{attribute 'qualified_only'}
{attribute 'strict'}
{attribute 'to_string'}
TYPE E_CollisionAvoidanceMode :
(
	SINGLE := 0,
	MULTI
);
END_TYPE

(* stored: Version 1.1.0.1
   DUT E_CollisionAvoidanceMode: Id {28e755ba-6279-4882-84f8-783382f25497} *)
